FUNCTION QUARTERS_TO_BYTE
  (* Standard: 61499-1 *)
  (* Version 1.0, 2024-02-22, franz *)
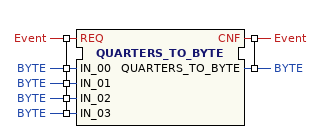
  EVENT_INPUT
    REQ WITH IN_00, IN_01, IN_02, IN_03;
  END_EVENT
  EVENT_OUTPUT
    CNF WITH QUARTERS_TO_BYTE;
  END_EVENT
  VAR_INPUT
    IN_00 : BYTE; (* QUARTER BYTE 00 *)
    IN_01 : BYTE; (* QUARTER BYTE 01 *)
    IN_02 : BYTE; (* QUARTER BYTE 02 *)
    IN_03 : BYTE; (* QUARTER BYTE 03 *)
  END_VAR
  VAR_OUTPUT
    QUARTERS_TO_BYTE : BYTE;
  END_VAR
  BODY IN ST:
FUNCTION QUARTERS_TO_BYTE : BYTE

VAR_INPUT
	IN_00 : BYTE;    // QUARTER BYTE 00
	IN_01 : BYTE;    // QUARTER BYTE 01
	IN_02 : BYTE;    // QUARTER BYTE 02
	IN_03 : BYTE;    // QUARTER BYTE 03
END_VAR

(* this Function combines the 4 QUARTER BYTES to a byte *)
QUARTERS_TO_BYTE := BYTE_QUARTER_ZZ;
QUARTERS_TO_BYTE := QUARTERS_TO_BYTE OR SHL(IN_03, SHFT_QUARTER_03);
QUARTERS_TO_BYTE := QUARTERS_TO_BYTE OR SHL(IN_02, SHFT_QUARTER_02);
QUARTERS_TO_BYTE := QUARTERS_TO_BYTE OR SHL(IN_01, SHFT_QUARTER_01);
QUARTERS_TO_BYTE := QUARTERS_TO_BYTE OR SHL(IN_00, SHFT_QUARTER_00);

END_FUNCTION
  END_BODY
END_FUNCTION
